Fanuc KAREL source: ko00007.KL

-- PROVISIONAL review KL for V1013-1; original PC SHA256 76e6a15d379c0465d5c3ffb03cfdf261fc66f269fee0acd072b1c3faf2f6223d
-- Incomplete behavior may be omitted. Consult companion uncertainty JSON. Do not deploy.
PROGRAM KO00007
%NOLOCKGROUP
-- UNRESOLVED_DECL P1 type=000101
-- UNRESOLVED_DECL P2 type=000101
-- UNRESOLVED_DECL P3 type=000101
-- UNRESOLVED_DECL P4 type=000101
-- UNRESOLVED_DECL OUT type=000106
BEGIN
  -- UNRESOLVED_PC offsets 5-68; opcodes 27,22,1C,22,1C,22,1C,22,1C,76,7E,4A
  -- UNRESOLVED_PC offsets 73-77; opcodes 7F
END KO00007
